{attribute 'qualified_only'}
VAR_GLOBAL
END_VAR

(* stored: Version 1.1.0.1
   GVL GVL_Variables: Id {5b2ad3d4-a585-0c6f-227f-c8cc96a9a687} *)
